Staubli VAL3: _sendStatus.pgx

program _sendStatus()
  local num l_nData
begin
  // ============================================================================
  // 상태 응답 전송 (1바이트)
  // 0=Idle, 1=Ready, 2=PassDone, 3=Error
  // ============================================================================

  l_nData = nStatusSignal
  sioSet(siTcpIpFbk, l_nData)

  putln("[TCP] STATUS = " + toString("", nStatusSignal))

end
